FUNCTION_BLOCK AirPiston
VAR_INPUT CONSTANT
	bEnable : BOOL;
END_VAR
VAR_OUTPUT
	valveExtend AT %Q* : BOOL;
	valveRetract AT %Q* : BOOL;
	
	contact AT %I* : BOOL;
	
	home AT %I* : BOOL;
	innerLimit AT %I* : BOOL;
	
	ready : BOOL;
	busy : BOOL;
	error : BOOL;
	homeSet : BOOL;
END_VAR
VAR
	reversalBrakeTrig : R_TRIG;
	brakePulse : TP;
	
	step : Homing;
	mode : (HOLD, IN, OUT);
END_VAR
VAR_STAT CONSTANT
	brakeTime : TIME := T#500MS;
END_VAR

IF NOT bEnable THEN
	valveExtend := FALSE;
	valveRetract := FALSE;
	RETURN;
END_IF

brakePulse(IN:= , PT:= brakeTime, Q=> , ET=> ); //reversal to act as brake
brakePulse.IN := brakePulse.IN AND brakePulse.Q; //automatically turn off pulse

IF home AND valveRetract THEN
	mode := HOLD;
ELSIF (innerLimit OR contact) AND valveExtend THEN
	brakePulse.IN := TRUE;
	mode := HOLD; //mode HOLD turns off valveExtend, so brakePulse timer is not started again
END_IF

CASE mode OF
	HOLD:
		valveExtend := FALSE;
		valveRetract := FALSE;
		
	IN:
		valveExtend := TRUE;
		valveRetract := FALSE;
		
	OUT:
		valveExtend := FALSE;
		valveRetract := TRUE;
		
END_CASE

valveRetract := valveRetract OR brakePulse.Q; //from mode or brake

METHOD extend : BOOL
VAR_INPUT
END_VAR
mode := IN;
END_METHOD

METHOD homingSequence : BOOL
(*
this version of homing always traverses to the inner limit before returning to home,
eliminating the possibility of reaching the outer limit while homing
*)
CASE step OF
	Homing.IDLE:
		step := Homing.HOME_OUT;
		
	Homing.REDO: //technically HOME_IN, towards travel limit
		mode := IN;
		valveExtend := TRUE;
		valveRetract := FALSE;
		
		IF innerLimit THEN
			valveExtend := FALSE;
			valveRetract := FALSE;
			step := Homing.HOME_OUT;
		END_IF
		
	Homing.HOME_OUT: //towards home
		mode := OUT;
		valveExtend := FALSE;
		valveRetract := TRUE;
		
		IF home THEN //if reached home
			valveExtend := FALSE;
			valveRetract := FALSE;
			step := Homing.DONE;
		END_IF
		
	Homing.DONE:
		mode := HOLD;
		valveExtend := FALSE;
		valveRetract := FALSE;
		homeSet := TRUE;
		
		homingSequence := TRUE;		
	
END_CASE
END_METHOD

METHOD retract : BOOL
VAR_INPUT
END_VAR
mode := OUT;
END_METHOD

METHOD stop : BOOL
VAR_INPUT
END_VAR
valveExtend := FALSE;
valveRetract := FALSE;
mode := HOLD;
END_METHOD

END_FUNCTION_BLOCK

(* stored: Version 1.1.0.1, ProductVersion 3.1.4024.11
   POU AirPiston: Id {ef8d0471-4ac2-4d12-9e08-c4e8a3719cb6}, SpecialFunc None
   Method extend: Id {c905417d-ebb0-4426-b712-8b35f4512697}
   Method homingSequence: Id {c3ff30f8-ced2-4f8e-b758-e21ca109ec69}
   Method retract: Id {d6cfbb92-1846-4f17-b88f-dcdab10c19f1}
   Method stop: Id {c035c442-83bc-4f21-a06c-19730e7f9f48} *)
